// TIA Portal V19 export
DATA_BLOCK "MODE SELECTION DB"   // DB3
{ S7_Optimized_Access := 'TRUE' }
// stored: MemoryReserve 100
   VAR
      AUTO : Bool;
      MANUAL : Bool;
      STANDBY : Bool;
   END_VAR
   VAR RETAIN
      "MODE BUFF" : Int;
      "PROCESS BUFF" : Int;
   END_VAR
BEGIN
END_DATA_BLOCK
